// :Description: Lives outside the solution directory; only reachable via the .sln reference.
FUNCTION_BLOCK FB_Remote
VAR
    counter : UDINT;
END_VAR


counter := counter + 1;

END_FUNCTION_BLOCK

(* stored: Version 1.1.0.1, ProductVersion 3.1.4026.0
   POU FB_Remote: Id {bbbbbbbb-bbbb-bbbb-bbbb-bbbbbbbbbbb1}, SpecialFunc None *)
